FUNCTION_BLOCK StopStart (* Composite Function Block Type *)
  (* Standard: 61499-2 *)
  (* Version 0.0, 7/14/2026, Schneider Electric, template *)
  PACKAGE SE.Nereda;
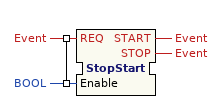
  EVENT_INPUT
    REQ WITH Enable; (* Normal Execution Request *)
  END_EVENT
  EVENT_OUTPUT
    START; (* Execution Confirmation *)
    STOP;
  END_EVENT
  VAR_INPUT
    Enable : BOOL; (* Input event qualifier *)
  END_VAR
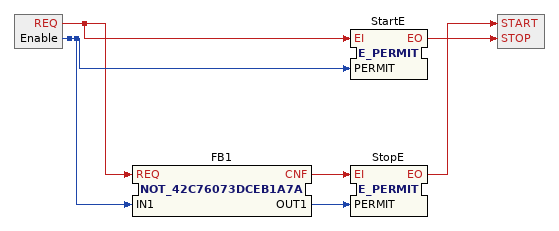
  FBS
    StartE : E_PERMIT;
    StopE : E_PERMIT;
    FB1 : NOT_42C76073DCEB1A7A; {SET_ATTRIBUTE(Configuration.GenericFBType.InterfaceParams, Runtime.Standard#CNT:=1;OUT${CNT$}:BOOL)}
  END_FBS
  EVENT_CONNECTIONS
    StartE.EO TO STOP;
    REQ TO StartE.EI;
    FB1.CNF TO StopE.EI;
    StopE.EO TO START;
    REQ TO FB1.REQ;
  END_CONNECTIONS
  DATA_CONNECTIONS
    Enable TO StartE.PERMIT;
    FB1.OUT1 TO StopE.PERMIT;
    Enable TO FB1.IN1;
  END_CONNECTIONS
END_FUNCTION_BLOCK
